INTERFACE ITcoServiceable

PROPERTY IsService : BOOL
GET
END_GET
END_PROPERTY

METHOD PUBLIC Service
END_METHOD

END_INTERFACE

(* stored: Version 1.1.0.1
   Itf ITcoServiceable: Id {226fd2d6-401e-4c29-97f4-f7e58b55d445}
   Property IsService: Id {d47aaea4-ce72-0454-0754-1e87b02cbd5e}
   Get Get: Id {d2b12008-0f0e-0a13-031e-805227a0361c}
   Method Service: Id {b2fe216f-37ab-46ad-9d62-c3f8870418e6} *)
